PROGRAM MAIN
VAR
    simRelay : SimRelay;
    simOven : SimOven;
END_VAR

simRelay();
simOven();

END_PROGRAM

(* stored: Version 1.1.0.1, ProductVersion 3.1.4024.4
   POU MAIN: Id {bda779b6-34ba-4438-8015-baa0f5e2c171}, SpecialFunc None *)
